FUNCTION_BLOCK FB_SEL_TIME (* TIME Selection *)
  (* Standard: 61499-1-D.1; Classification: Selection Functions *)
  (* Version 0.1, 2001-08-06, JHC, Rockwell Automation, XML version *)
  (* Version 0.0, 1999-02-19, JHC, Rockwell Automation, SRC version *)
  (* Compiler header: package fb.rt.math; *)
  (* Compiler classdef: class FB_SEL_TIME extends FBSelectFunction *)
  (* Compiler Java IBM VisualAge 3.0 *)
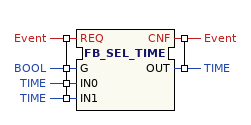
  EVENT_INPUT
    REQ WITH G, IN0, IN1;
  END_EVENT
  EVENT_OUTPUT
    CNF WITH OUT;
  END_EVENT
  VAR_INPUT
    G : BOOL; (* Selector *)
    IN0 : TIME; (* Selected when G=0 *)
    IN1 : TIME; (* Selected when G=1 *)
  END_VAR
  VAR_OUTPUT
    OUT : TIME; (* Selected value *)
  END_VAR
END_FUNCTION_BLOCK
